FUNCTION_BLOCK WriteLRealIf
VAR_IN_OUT
	Out: LREAL;
END_VAR
VAR_INPUT
	EN: BOOL := TRUE;
	In: LREAL;
END_VAR
VAR_OUTPUT
	ENO: bool;
END_VAR
VAR
END_VAR

ENO := EN;
IF EN THEN
	Out := In;
ELSE
	Out := 0.0;	
END_IF

END_FUNCTION_BLOCK

(* stored: Version 1.1.0.1, ProductVersion 3.1.4024.6
   POU WriteLRealIf: Id {c4c78d15-a769-439d-aef5-fe9424c9b94e}, SpecialFunc None *)
